// TIA Portal V19 export
FUNCTION "Polygon Monitoring" : Void   // FC111, FBD
TITLE = Polygon - Process Monitoring
{ S7_Optimized_Access := 'TRUE' }
// stored: AutoNumber false, SetENOAutomatically false
   VAR_TEMP
      tmp : Bool;
      HT_reset : Real;
      LT_Reset : Real;
      deadband : Real;
   END_VAR
   VAR_TEMP   // added for the SCL form of the ladder/FBD networks
      _w1 : Bool;
      _s5time1 : S5Time;
      _w2 : Bool;
      _s5time2 : S5Time;
   END_VAR
BEGIN

NETWORK
TITLE = Condenstate deadbands
      L     3.0;
      T     #deadband;
      L     "Setpoints_Polygon".TT0941_CondenseHigh;
      L     #deadband;
      -R;
      T     #HT_reset;
      L     "Setpoints_Polygon".TT0941_CondenseLow;
      L     #deadband;
      +R;
      T     #LT_Reset;



NETWORK
TITLE = TT0941 Condensate temperature High or Low
// Allow condensate temperature to attain temperature from cold start and 
// stabilise after 3 bar steam.
      A(;
      O(;
      L     "PG_Devices".TTX0941.Value;
      L     "Setpoints_Polygon".TT0941_CondenseHigh;
      >R;
      );
      O(;
      L     "PG_Devices".TTX0941.Value;
      L     "Setpoints_Polygon".TT0941_CondenseLow;
      <R;
      );
      );
      R     "M21.2";
      A(;
      O(;
      L     "PG_Devices".TTX0941.Value;
      L     #LT_Reset;
      >R;
      );
      A(;
      L     "PG_Devices".TTX0941.Value;
      L     #HT_reset;
      <R;
      );
      );
      S     "M21.2";
      AN    "M21.2";
      A(;
      A     "PG_Devices".V0935.IN.Activate;
      AN    "PG_Devices".V0552.IN.Activate;
      L     S5T#10M;
      SD    "Tag_111";
      NOP   0;
      NOP   0;
      NOP   0;
      A     "Tag_111";
      );
      S     "ProcessAndPbAlarms"."A"[69];  //A69_TT0941_TempFault


REGION Network 3: TT0940 temperature Low
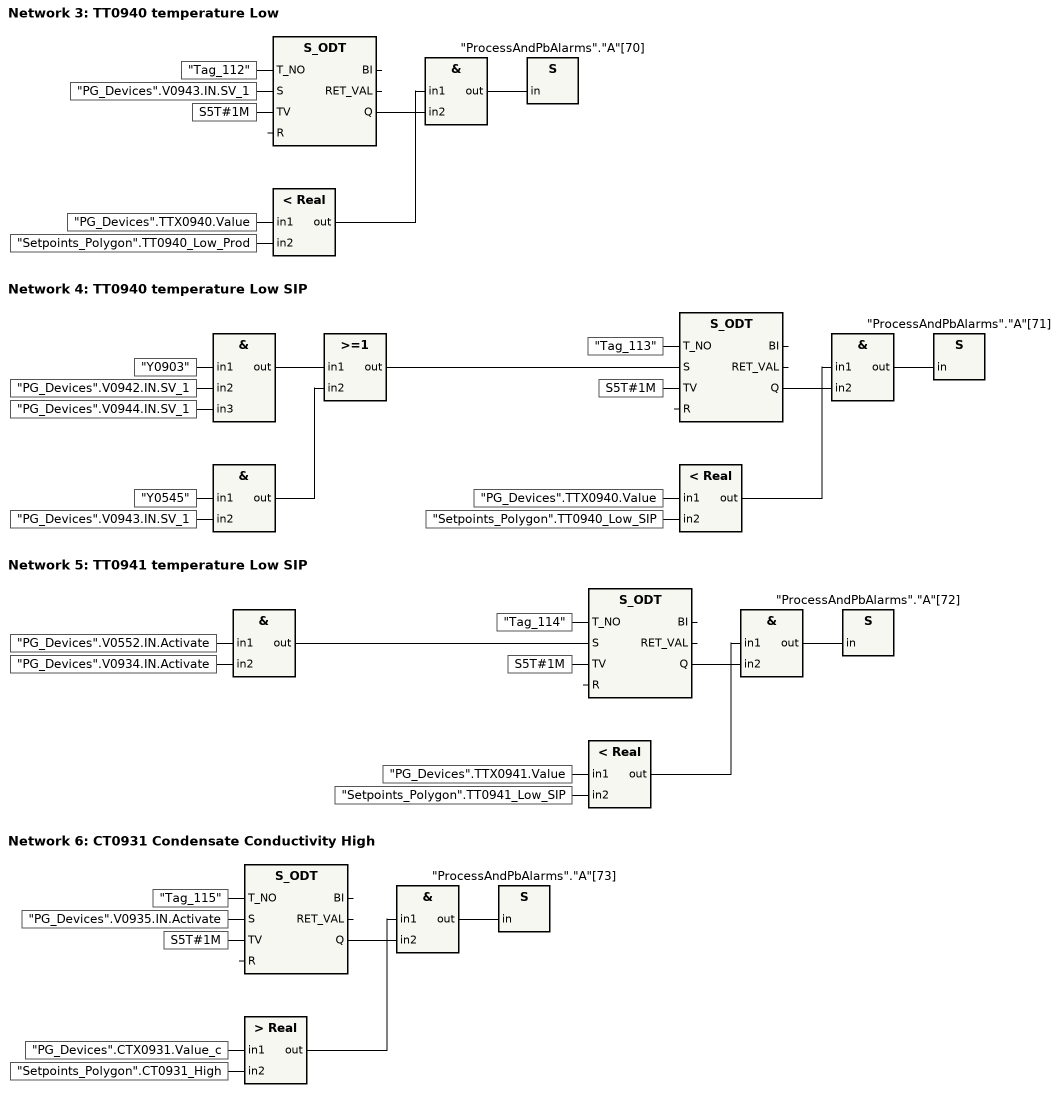
   #_s5time1 := S_ODT(T_NO := "Tag_112", S := "PG_Devices".V0943.IN.SV_1, TV := S5T#1M, Q => #_w1);
   IF ("PG_Devices".TTX0940.Value < "Setpoints_Polygon".TT0940_Low_Prod) AND #_w1 THEN
       "ProcessAndPbAlarms"."A"[70] := TRUE;
   END_IF;
END_REGION

REGION Network 4: TT0940 temperature Low SIP
   #_s5time1 := S_ODT(T_NO := "Tag_113",
                      S := ("Y0903" AND "PG_Devices".V0942.IN.SV_1 AND "PG_Devices".V0944.IN.SV_1) OR ("Y0545" AND "PG_Devices".V0943.IN.SV_1),
                      TV := S5T#1M,
                      Q => #_w1);
   IF ("PG_Devices".TTX0940.Value < "Setpoints_Polygon".TT0940_Low_SIP) AND #_w1 THEN
       "ProcessAndPbAlarms"."A"[71] := TRUE;
   END_IF;
END_REGION

REGION Network 5: TT0941 temperature Low SIP
   #_s5time1 := S_ODT(T_NO := "Tag_114",
                      S := "PG_Devices".V0552.IN.Activate AND "PG_Devices".V0934.IN.Activate,
                      TV := S5T#1M,
                      Q => #_w1);
   IF ("PG_Devices".TTX0941.Value < "Setpoints_Polygon".TT0941_Low_SIP) AND #_w1 THEN
       "ProcessAndPbAlarms"."A"[72] := TRUE;
   END_IF;
END_REGION

REGION Network 6: CT0931 Condensate Conductivity High
   #_s5time1 := S_ODT(T_NO := "Tag_115", S := "PG_Devices".V0935.IN.Activate, TV := S5T#1M, Q => #_w1);
   IF ("PG_Devices".CTX0931.Value_c > "Setpoints_Polygon".CT0931_High) AND #_w1 THEN
       "ProcessAndPbAlarms"."A"[73] := TRUE;
   END_IF;
END_REGION

NETWORK
TITLE = EOL temperature Low Production
      A(;
      L     "PG_Devices".TTX1040.Value;
      L     "Setpoints_Polygon".EOL_Barrier_Low_Prod;
      <R;
      );
      O(;
      L     "PG_Devices".TTX1041.Value;
      L     "Setpoints_Polygon".EOL_Barrier_Low_Prod;
      <R;
      );
      A(;
      A     "PG_Devices".V1024.IN.Activate;
      L     S5T#1M;
      SD    "Tag_116";
      NOP   0;
      NOP   0;
      NOP   0;
      A     "Tag_116";
      );
      S     "ProcessAndPbAlarms"."A"[74];

NETWORK
TITLE = EOL temperature Low SIP
      A(;
      L     "PG_Devices".TTX1040.Value;
      L     "Setpoints_Polygon".EOL_Barrier_Low_SIP;
      <R;
      );
      O(;
      L     "PG_Devices".TTX1041.Value;
      L     "Setpoints_Polygon".EOL_Barrier_Low_SIP;
      <R;
      );
      A(;
      AN    "PG_Devices".V1024.IN.Activate;
      A     "MY0903";
      A     "PG_Devices".V1021.IN_SV_1;
      L     S5T#1M;
      SD    "Tag_117";
      NOP   0;
      NOP   0;
      NOP   0;
      A     "Tag_117";
      );
      S     "ProcessAndPbAlarms"."A"[75];

REGION Network 9: SIP - High Temperature warning alarm
   // Triggered, if any PG Transfer Line TTx above 140C
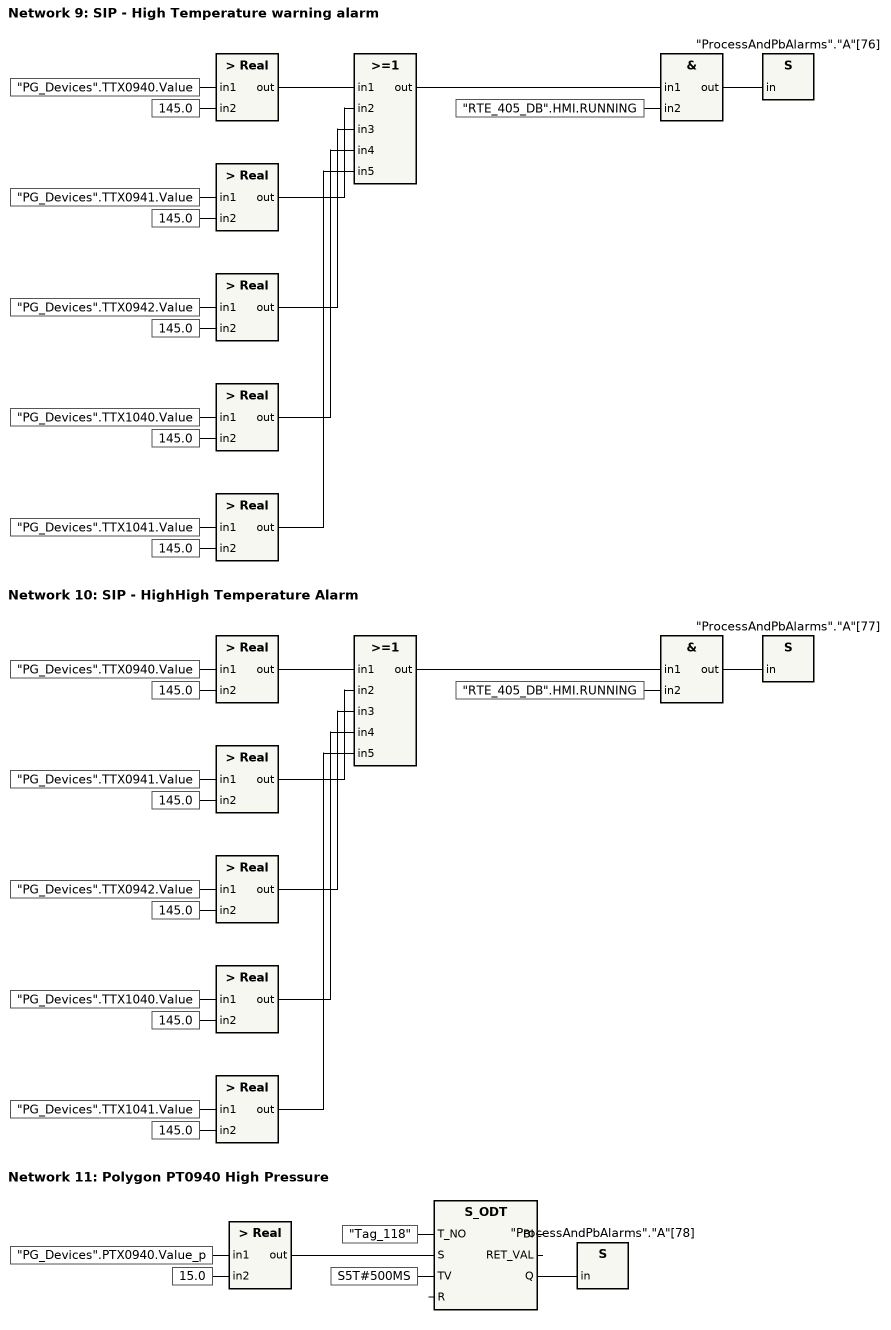
   IF (("PG_Devices".TTX0940.Value > 145.0) OR ("PG_Devices".TTX0941.Value > 145.0) OR ("PG_Devices".TTX0942.Value > 145.0) OR ("PG_Devices".TTX1040.Value > 145.0) OR ("PG_Devices".TTX1041.Value > 145.0)) AND "RTE_405_DB".HMI.RUNNING THEN
       "ProcessAndPbAlarms"."A"[76] := TRUE;
   END_IF;
END_REGION

REGION Network 10: SIP - HighHigh Temperature Alarm
   // Triggered, if any PG Transfer Line TTx above 145C and Auto Abort SIP
   IF (("PG_Devices".TTX0940.Value > 145.0) OR ("PG_Devices".TTX0941.Value > 145.0) OR ("PG_Devices".TTX0942.Value > 145.0) OR ("PG_Devices".TTX1040.Value > 145.0) OR ("PG_Devices".TTX1041.Value > 145.0)) AND "RTE_405_DB".HMI.RUNNING THEN
       "ProcessAndPbAlarms"."A"[77] := TRUE;
   END_IF;
END_REGION

REGION Network 11: Polygon PT0940 High Pressure
   // Set PTX0940 High Pressure Alarm at 15 bar
   #_s5time1 := S_ODT(T_NO := "Tag_118", S := "PG_Devices".PTX0940.Value_p > 15.0, TV := S5T#500MS, Q => #_w1);
   IF #_w1 THEN "ProcessAndPbAlarms"."A"[78] := TRUE; END_IF;
END_REGION

REGION Network 12: CTX22.74 - Polygon Filler 2 - Product at Filler
   // Signal to Fruit Plant Alsafe  I 41.2
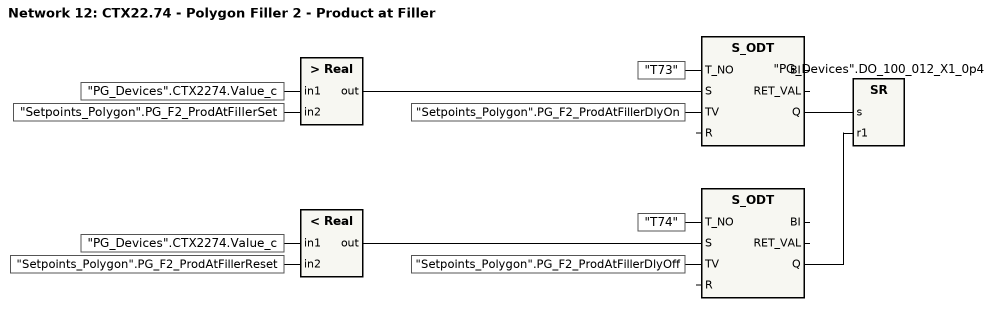
   #_s5time1 := S_ODT(T_NO := "T73",
                      S := "PG_Devices".CTX2274.Value_c > "Setpoints_Polygon".PG_F2_ProdAtFillerSet,
                      TV := "Setpoints_Polygon".PG_F2_ProdAtFillerDlyOn,
                      Q => #_w1);
   #_s5time2 := S_ODT(T_NO := "T74",
                      S := "PG_Devices".CTX2274.Value_c < "Setpoints_Polygon".PG_F2_ProdAtFillerReset,
                      TV := "Setpoints_Polygon".PG_F2_ProdAtFillerDlyOff,
                      Q => #_w2);
   IF #_w1 THEN
       "PG_Devices".DO_100_012_X1_0p4 := TRUE;   // SR flip-flop
   END_IF;
   IF #_w2 THEN "PG_Devices".DO_100_012_X1_0p4 := FALSE; END_IF;
END_REGION
END_FUNCTION
